INTERFACE ITF_Motor_1

PROPERTY ActualState : BOOL
GET
END_GET
END_PROPERTY

METHOD Auto : BOOL
VAR_INPUT
END_VAR
END_METHOD

PROPERTY Error_State : BOOL
GET
END_GET
END_PROPERTY

METHOD Manueel : BOOL
VAR_INPUT
END_VAR
END_METHOD

METHOD Reset : BOOL
VAR_INPUT
END_VAR
END_METHOD

METHOD Richting_L : BOOL
VAR_INPUT
END_VAR
END_METHOD

METHOD Richting_R : BOOL
VAR_INPUT
END_VAR
END_METHOD

METHOD Start : BOOL
VAR_INPUT
END_VAR
END_METHOD

PROPERTY State : E_MotorState
GET
END_GET
END_PROPERTY

METHOD Stop : BOOL
VAR_INPUT
END_VAR
END_METHOD

METHOD Toerental : INT
VAR_INPUT
END_VAR
END_METHOD

END_INTERFACE

(* stored: Version 1.1.0.1, ProductVersion 3.1.4024.12
   Itf ITF_Motor_1: Id {91bb75c3-0eea-4948-b6fa-d22d45de9de0}
   Folder Methods: Id {05cee666-7261-4506-bd42-a9d3e1ab907a}
   Folder Properties: Id {5a756104-037d-4f39-a817-efae77a47e69}
   Property ActualState: Id {58b8f85d-fc8b-4544-9814-7c31c51d4939}
   Get Get: Id {d6280de5-71b7-4f26-bb86-df6a1dc71dcb}
   Method Auto: Id {76858ff0-4fd4-4320-9110-a8cb056b9886}
   Property Error_State: Id {b7650939-7fff-480c-b9e7-b0b9cae6b7f3}
   Get Get: Id {169b7ccb-be68-4d65-8b31-e60bb6dbe9cc}
   Method Manueel: Id {17131916-26de-44cf-9ae6-c2754302f543}
   Method Reset: Id {b2a15614-ce49-4830-a720-02ee7a2c8817}
   Method Richting_L: Id {205a2fef-aeb9-4f68-9709-b96623a1a811}
   Method Richting_R: Id {6dafc7ba-7ae0-405b-96d7-2ff49a93af2f}
   Method Start: Id {f75b733a-46db-488f-b841-f282967d6767}
   Property State: Id {f0747509-035d-4046-baf2-317499555aed}
   Get Get: Id {9f8f106c-c395-498c-9159-e8e5c6a43cf6}
   Method Stop: Id {c25481e4-264d-47ce-8f03-3321d497d4a1}
   Method Toerental: Id {910f9299-17ed-41a5-9b54-8c39c72b44de} *)
